FUNCTION_BLOCK BistableCylinder EXTENDS BaseCylinder
VAR_INPUT	
END_VAR
VAR_OUTPUT
END_VAR
VAR	
	//Hardware
	DO_Retract AT %Q* : BOOL;
END_VAR

METHOD METH_Extend : BOOL
DO_Extend := TRUE;
DO_Retract := FALSE;
END_METHOD

METHOD METH_Retract : BOOL
DO_Extend := FALSE;
DO_Retract := TRUE;
END_METHOD

END_FUNCTION_BLOCK

(* stored: Version 1.1.0.1, ProductVersion 3.1.4024.9
   POU BistableCylinder: Id {d2153795-1ca1-44de-a399-9e53c1075eb0}, SpecialFunc None
   Method METH_Extend: Id {c672904d-c1ad-46b0-91d7-b77b03bd09c4}
   Method METH_Retract: Id {3167b7ec-5429-406b-a4ac-69c28dcd1bf7} *)
